// TwinCAT 3 PLC project tcl_Utilities
// Title: tcl_Utilities
// Company: Red Rock Controls Limited
// Author: Roger Christopher
// ProjectVersion: 1.0.9.0
// Description: F_LogError, etc added tcl_EventLog lib ref removed
// ProgramVersion: 3.1.4023.0
// libraries:
//   Tc2_Standard, * (Beckhoff Automation GmbH)
//   Tc2_System, * (Beckhoff Automation GmbH)
//   Tc2_Utilities, * (Beckhoff Automation GmbH)
//   Tc3_Module, * (Beckhoff Automation GmbH)
//   tcl_Events, * (Red Rock Controls Limited)
//   tcl_Execution, * (Red Rock Controls Limited)
//   tcl_UnitTest, * (Red Rock Controls Limited)
// project tree:
//   Classes/Clock/Event Definitions/Day Changed/ IEventHandler_OnDayChanged.TcIO, TEvent_DayChanged.TcPOU
//   Classes/Clock/Event Definitions/Hours Changed/ IEventHandler_OnHourChanged.TcIO, TEvent_HoursChanged.TcPOU
//   Classes/Clock/Event Definitions/Minutes Changed/ IEventHandler_OnMinutesChanged.TcIO, TEvent_MinutesChanged.TcPOU
//   Classes/Clock/Event Definitions/Seconds Changed/ IEventHandler_OnSecondsChanged.TcIO, TEvent_SecondsChanged.TcPOU
//   Classes/Clock/ IClock.TcIO, TClock.TcPOU, TClockEventSource.TcPOU
//   Classes/Edge Detection/ TFallingEdge.TcPOU (not stored), TRisingEdge.TcPOU
//   Classes/Licence Check/ TLicenceCheck.TcPOU
//   Classes/Misc/ TCounter.TcPOU, TCsvString.TcPOU, TGetTimeZoneInfo.TcPOU, TRestartTwinCAT.TcPOU, TRingCounter_INT.TcPOU, TRingCounter_UDINT.TcPOU, TRollingAverage.TcPOU, TSetWindowsClock.TcPOU, TShutdown.TcPOU, TStartProcess.TcPOU
//   Classes/String Split/ TStringSplitter.TcPOU (not stored)
//   Classes/Timers/ TOffTimer.TcPOU (not stored), TOnTimer.TcPOU, TPulseTimer.TcPOU
//   Classes/Value Monitor/ TValueMonitor.TcPOU, TValueMonitorEx.TcPOU
//   Function Blocks/ FB_AutoReset.TcPOU, FB_ValueChanged.TcPOU
//   Functions/Date Time Formatting/ F_DateAsString.TcPOU, F_DateTimeAsString.TcPOU, F_DateTimeAsString_ms.TcPOU, F_TimeAsString.TcPOU, F_TimeAsString_ms.TcPOU, F_TimestampAsFilenameString.TcPOU (not stored)
//   Functions/Event Logging/ F_LogError.TcPOU, F_LogMessage.TcPOU, F_LogWarning.TcPOU
//   Functions/General/ F_ClearMem.TcPOU (not stored), F_GetAdsPort.TcPOU (not stored)
//   Functions/Misc/ F_Assert.TcPOU (not stored), F_Equals.TcPOU (not stored)
//   Functions/String Formatting/ F_FormatString1.TcPOU (not stored), F_FormatString10.TcPOU (not stored), F_FormatString2.TcPOU (not stored), F_FormatString3.TcPOU (not stored), F_FormatString4.TcPOU (not stored), F_FormatString5.TcPOU, F_FormatString6.TcPOU (not stored), F_FormatString7.TcPOU (not stored), F_FormatString8.TcPOU (not stored), F_FormatStringEx1.TcPOU (not stored), F_FormatStringEx10.TcPOU, F_FormatStringEx2.TcPOU (not stored), F_FormatStringEx3.TcPOU (not stored), F_FormatStringEx4.TcPOU (not stored), F_FormatStringEx5.TcPOU (not stored), F_FormatStringEx6.TcPOU, F_FormatStringEx7.TcPOU (not stored), F_FormatStringEx8.TcPOU, F_LREAL_TO_STRING.TcPOU (not stored), F_LTrimEx.TcPOU (not stored), F_PadString.TcPOU, F_RTrimEx.TcPOU, F_STRING_TO_ARG.TcPOU (not stored), F_Trim.TcPOU (not stored)
//   / GlobalTextList.TcGTLO (not stored), Param.TcGVL, PlcTask.TcTTO, Visualization Manager.TcVMO (not stored)
//   Unit Tests/Clock/ Test_Raises_OnDaysChanged.TcPOU, Test_Raises_OnHoursChanged.TcPOU, Test_Raises_OnMinutesChanged.TcPOU, Test_Raises_OnSecondsChanged.TcPOU
//   Unit Tests/Date Time Formatting Tests/ Test_DateAsString.TcPOU, Test_DateTimeAsString.TcPOU, Test_DateTimeAsString_ms.TcPOU, Test_TimeAsString_24HourFormat.TcPOU, Test_TimeAsString_IncludesLeadingZeros.TcPOU, Test_TimestampAsFilenameString.TcPOU, Test_TimeAsString_ms.TcPOU
//   Unit Tests/Licence Check/ Test_LicenceCheck_GetsInValidLicence.TcPOU, Test_LicenceCheck_GetsValidLicence.TcPOU
//   Unit Tests/ PB_TestRunner.TcPOU
//   Unit Tests/String Split/ Test_StringSplitter_Handles_Empty_String.TcPOU, Test_StringSplitter_ReturnsRemainder.TcPOU, Test_StringSplitter_Splits_On_Tab.TcPOU
//   Version/ Global_Version.TcGVL
//   Visualisation/ Visualization.TcVIS
// real-time tasks:
//   TASK PlcTask: cycle T#10ms, priority 20, ADS port 350

CONFIGURATION tcl_Utilities
    RESOURCE PLC ON TwinCAT3
        TASK PlcTask(INTERVAL := T#10ms, PRIORITY := 20);
        PROGRAM PB_TestRunner WITH PlcTask : PB_TestRunner;
    END_RESOURCE
END_CONFIGURATION

// ---- Param.TcGVL
{attribute 'qualified_only'}
VAR_GLOBAL CONSTANT
    MaxCsvFields : INT := 99;
END_VAR

// ---- Version/Global_Version.TcGVL
{attribute 'TcGenerated'}
{attribute 'no-analysis'}
{attribute 'linkalways'}
// This function has been automatically generated from the project information.
VAR_GLOBAL CONSTANT
	{attribute 'const_non_replaced'}
	stLibVersion_tcl_Utilities : ST_LibVersion := (iMajor := 1, iMinor := 0, iBuild := 9, iRevision := 0, nFlags := 0, sVersion := '1.0.9.0');
END_VAR

// ---- Classes/Clock/Event Definitions/Day Changed/IEventHandler_OnDayChanged.TcIO
INTERFACE IEventHandler_OnDayChanged EXTENDS IEventHandlerBase

METHOD OnDayChanged
VAR_INPUT
	Now: TIMESTRUCT;
END_VAR
END_METHOD

END_INTERFACE

// ---- Classes/Clock/Event Definitions/Hours Changed/IEventHandler_OnHourChanged.TcIO
INTERFACE IEventHandler_OnHourChanged EXTENDS IEventHandlerBase

METHOD OnHourChanged
VAR_INPUT
	Now: TIMESTRUCT;
END_VAR
END_METHOD

END_INTERFACE

// ---- Classes/Clock/Event Definitions/Minutes Changed/IEventHandler_OnMinutesChanged.TcIO
INTERFACE IEventHandler_OnMinutesChanged EXTENDS IEventHandlerBase

METHOD OnMinutesChanged
VAR_INPUT
	Now: TIMESTRUCT;
END_VAR
END_METHOD

END_INTERFACE

// ---- Classes/Clock/Event Definitions/Seconds Changed/IEventHandler_OnSecondsChanged.TcIO
INTERFACE IEventHandler_OnSecondsChanged EXTENDS IEventHandlerBase

METHOD OnSecondsChanged
VAR_INPUT
	Now: TIMESTRUCT;
END_VAR
END_METHOD

END_INTERFACE

// ---- Classes/Clock/IClock.TcIO
INTERFACE IClock

PROPERTY DateTimeInitialised : BOOL
GET
END_GET
END_PROPERTY

PROPERTY NowAsDateTime : DT
GET
END_GET
END_PROPERTY

PROPERTY NowAsTimeStruct : REFERENCE TO TIMESTRUCT
GET
END_GET
END_PROPERTY

END_INTERFACE

// ---- Unit Tests/PB_TestRunner.TcPOU
PROGRAM PB_TestRunner 
VAR
//    EnableAdsLogMessages_State : BOOL;
//    EnableAdsLogMessages_DuringTest : BOOL := FALSE; // inhibit Invalid Event Handler error message - confusing here
//    RisingEdge_TestsRunning  : TRisingEdge;
//    FallingEdge_TestsRunning : TFallingEdge;
    
    Test_Raises_OnDaysChanged                : Test_Raises_OnDaysChanged;
    Test_Raises_OnHoursChanged               : Test_Raises_OnHoursChanged;
    Test_Raises_OnMinutesChanged             : Test_Raises_OnMinutesChanged;
    Test_Raises_OnSecondsChanged             : Test_Raises_OnSecondsChanged;
                                             
    Test_DateAsString                        : Test_DateAsString;
    Test_DateTimeAsString                    : Test_DateTimeAsString;
    Test_DateTimeAsString_ms                 : Test_DateTimeAsString_ms;
    Test_TimeAsString_24HourFormat           : Test_TimeAsString_24HourFormat;
    Test_TimeAsString_IncludesLeadingZeros   : Test_TimeAsString_IncludesLeadingZeros;
    Test_TimeAsString_ms                     : Test_TimeAsString_ms;
    Test_TimestampAsFilenameString           : Test_TimestampAsFilenameString;
                                             
    Test_LicenceCheck_GetsInValidLicence     : Test_LicenceCheck_GetsInValidLicence;
    Test_LicenceCheck_GetsValidLicence       : Test_LicenceCheck_GetsValidLicence;
   
    Test_StringSplitter_Handles_Empty_String : Test_StringSplitter_Handles_Empty_String;
    Test_StringSplitter_ReturnsRemainder     : Test_StringSplitter_ReturnsRemainder;
    Test_StringSplitter_Splits_On_Tab        : Test_StringSplitter_Splits_On_Tab;

 
END_VAR

tcl_UnitTest.TestFramework.TestRunner();

//IF RisingEdge_TestsRunning.Test(tcl_UnitTest.UnitTests.TestFramework.TestsRunning) THEN
//    EnableAdsLogMessages_State := tcl_EventLog.EventLog.EnableAdsLogMessages; // store so we can restore previous state
//    EventLog.EnableAdsLogMessages := EnableAdsLogMessages_DuringTest;  // force the visibility of ads log messages
//END_IF

//IF FallingEdge_TestsRunning.Test(tcl_UnitTest.UnitTests.TestFramework.TestsRunning) THEN
//    EventLog.EnableAdsLogMessages := EnableAdsLogMessages_State; // restore previous state
//END_IF

END_PROGRAM

// ---- Unit Tests/Clock/Test_Raises_OnDaysChanged.TcPOU
FUNCTION_BLOCK Test_Raises_OnDaysChanged EXTENDS TUnitTestBase
IMPLEMENTS 
    IEventHandler_OnDayChanged
VAR
    NowFromEvent : TIMESTRUCT;
    
    OnDaysChanged_Raised    : BOOL;
END_VAR

METHOD  Execute
VAR_INST
    ClockEventSource : TClockEventSource;
    Now              : TIMESTRUCT := (wDay := 23, wMonth := 12, wYear := 1945, wHour := 22, wMinute := 20, wSecond := 18);
    OneDayLater      : TIMESTRUCT := (wDay := 24, wMonth := 12, wYear := 1945, wHour := 22, wMinute := 20, wSecond := 18);
END_VAR
OnDaysChanged_Raised := FALSE;

ClockEventSource.Event_DayChanged.ClearEventHandlers().AddEventHandler(THIS^);

ClockEventSource.Init(Now := Now);
ClockEventSource(Now := OneDayLater);

Assertion.AssertEquals_BOOL(
    Expected := TRUE,
    Actual   := OnDaysChanged_Raised,
    ObjectName := _TestName,
    VariableName  := 'OnDaysChanged_Raised');

Assertion.AssertEquals_STRUCT(
    Expected := OneDayLater,
    Actual   := NowFromEvent,
    ObjectName := _TestName,
    VariableName  := 'NowFromEvent');

Test_Finished();
END_METHOD

METHOD OnDayChanged
VAR_INPUT
	Now	: Tc2_Utilities.TIMESTRUCT;
END_VAR
NowFromEvent := Now;
OnDaysChanged_Raised := TRUE;
END_METHOD

END_FUNCTION_BLOCK

// ---- Classes/Clock/TClockEventSource.TcPOU
FUNCTION_BLOCK TClockEventSource
VAR_INPUT
    Now : TIMESTRUCT;
END_VAR
VAR
    _LastTickNowAsTimestruct : TIMESTRUCT;

    _Event_SecondsChanged : TEvent_SecondsChanged;
    _Event_MinutesChanged : TEvent_MinutesChanged;
    _Event_HoursChanged   : TEvent_HoursChanged;
    _Event_DayChanged     : TEvent_DayChanged;

END_VAR

IF Now.wSecond <> _LastTickNowAsTimestruct.wSecond THEN
    _Event_SecondsChanged.RaiseEx(Now);
END_IF
IF Now.wMinute <> _LastTickNowAsTimestruct.wMinute THEN
    _Event_MinutesChanged.RaiseEx(Now);
END_IF
IF Now.wHour <> _LastTickNowAsTimestruct.wHour THEN
    _Event_HoursChanged.RaiseEx(Now);
END_IF
IF Now.wDay <> _LastTickNowAsTimestruct.wDay THEN
    _Event_DayChanged.RaiseEx(Now);
END_IF

_LastTickNowAsTimestruct := Now;

PROPERTY Event_DayChanged : IEvent
GET
Event_DayChanged := _Event_DayChanged;
END_GET
END_PROPERTY

PROPERTY Event_HoursChanged : IEvent
GET
Event_HoursChanged := _Event_HoursChanged;
END_GET
END_PROPERTY

PROPERTY Event_MinutesChanged : IEvent
GET
Event_MinutesChanged := _Event_MinutesChanged;
END_GET
END_PROPERTY

PROPERTY Event_SecondsChanged : IEvent
GET
Event_SecondsChanged := _Event_SecondsChanged;
END_GET
END_PROPERTY

METHOD Init // initialise stored value so event handlers do not fire erroneously on first update
VAR_INPUT
    Now : TIMESTRUCT;
END_VAR
_LastTickNowAsTimestruct := Now;
END_METHOD

END_FUNCTION_BLOCK

// ---- Classes/Clock/Event Definitions/Seconds Changed/TEvent_SecondsChanged.TcPOU
FUNCTION_BLOCK TEvent_SecondsChanged EXTENDS TEventBase IMPLEMENTS IEvent
VAR
	Now: TIMESTRUCT;
    Handler : IEventHandler_OnSecondsChanged;
END_VAR

METHOD  CallHandler
VAR_INPUT
    HandlerBase : IEventHandlerBase;
END_VAR
IF __QUERYINTERFACE(HandlerBase,Handler) THEN
    Handler.OnSecondsChanged(Now);
END_IF
END_METHOD

METHOD  IsHandlerSupported : BOOL
VAR_INPUT
    EventHandler : IEventHandlerBase;
END_VAR
IF __QUERYINTERFACE(EventHandler,Handler) THEN
    IsHandlerSupported := TRUE;
END_IF
END_METHOD

METHOD RaiseEx
VAR_INPUT
	Now: TIMESTRUCT;
END_VAR
THIS^.Now := Now;
SUPER^.Raise();
END_METHOD

END_FUNCTION_BLOCK

// ---- Classes/Clock/Event Definitions/Minutes Changed/TEvent_MinutesChanged.TcPOU
FUNCTION_BLOCK TEvent_MinutesChanged EXTENDS TEventBase IMPLEMENTS IEvent
VAR
	Now: TIMESTRUCT;
    Handler : IEventHandler_OnMinutesChanged;
END_VAR

METHOD  CallHandler
VAR_INPUT
    HandlerBase : IEventHandlerBase;
END_VAR
IF __QUERYINTERFACE(HandlerBase,Handler) THEN
    Handler.OnMinutesChanged(Now);
END_IF
END_METHOD

METHOD  IsHandlerSupported : BOOL
VAR_INPUT
    EventHandler : IEventHandlerBase;
END_VAR
IF __QUERYINTERFACE(EventHandler,Handler) THEN
    IsHandlerSupported := TRUE;
END_IF
END_METHOD

METHOD RaiseEx
VAR_INPUT
	Now: TIMESTRUCT;
END_VAR
THIS^.Now := Now;
SUPER^.Raise();
END_METHOD

END_FUNCTION_BLOCK

// ---- Classes/Clock/Event Definitions/Hours Changed/TEvent_HoursChanged.TcPOU
FUNCTION_BLOCK TEvent_HoursChanged EXTENDS TEventBase IMPLEMENTS IEvent
VAR
	Now: TIMESTRUCT;
    Handler : IEventHandler_OnHourChanged;
END_VAR

METHOD  CallHandler
VAR_INPUT
    HandlerBase : IEventHandlerBase;
END_VAR
IF __QUERYINTERFACE(HandlerBase,Handler) THEN
    Handler.OnHourChanged(Now);
END_IF
END_METHOD

METHOD  IsHandlerSupported : BOOL
VAR_INPUT
    EventHandler : IEventHandlerBase;
END_VAR
IF __QUERYINTERFACE(EventHandler,Handler) THEN
    IsHandlerSupported := TRUE;
END_IF
END_METHOD

METHOD RaiseEx
VAR_INPUT
	Now: TIMESTRUCT;
END_VAR
THIS^.Now := Now;
SUPER^.Raise();
END_METHOD

END_FUNCTION_BLOCK

// ---- Classes/Clock/Event Definitions/Day Changed/TEvent_DayChanged.TcPOU
FUNCTION_BLOCK TEvent_DayChanged EXTENDS TEventBase IMPLEMENTS IEvent
VAR
	Now: TIMESTRUCT;
    Handler : IEventHandler_OnDayChanged;
END_VAR

METHOD  CallHandler
VAR_INPUT
    HandlerBase : IEventHandlerBase;
END_VAR
IF __QUERYINTERFACE(HandlerBase,Handler) THEN
    Handler.OnDayChanged(Now);
END_IF
END_METHOD

METHOD  IsHandlerSupported : BOOL
VAR_INPUT
    EventHandler : IEventHandlerBase;
END_VAR
IF __QUERYINTERFACE(EventHandler,Handler) THEN
    IsHandlerSupported := TRUE;
END_IF
END_METHOD

METHOD RaiseEx
VAR_INPUT
	Now: TIMESTRUCT;
END_VAR
THIS^.Now := Now;
SUPER^.Raise();
END_METHOD

END_FUNCTION_BLOCK

// ---- Unit Tests/Clock/Test_Raises_OnHoursChanged.TcPOU
FUNCTION_BLOCK Test_Raises_OnHoursChanged EXTENDS TUnitTestBase
IMPLEMENTS 
    IEventHandler_OnHourChanged
VAR
    NowFromEvent : TIMESTRUCT;
    
    OnHoursChanged_Raised    : BOOL;
END_VAR

METHOD  Execute
VAR_INST
    ClockEventSource : TClockEventSource;
    Now              : TIMESTRUCT := (wDay := 23, wMonth := 12, wYear := 1945, wHour := 22, wMinute := 20, wSecond := 18);
    OneHourLater     : TIMESTRUCT := (wDay := 23, wMonth := 12, wYear := 1945, wHour := 23, wMinute := 20, wSecond := 18);
END_VAR
OnHoursChanged_Raised := FALSE;

ClockEventSource.Event_HoursChanged.ClearEventHandlers().AddEventHandler(THIS^);

ClockEventSource.Init(Now := Now);
ClockEventSource(Now := OneHourLater);

Assertion.AssertEquals_BOOL(
    Expected := TRUE,
    Actual   := OnHoursChanged_Raised,
    ObjectName := _TestName,
    VariableName  := 'OnHoursChanged_Raised');

Assertion.AssertEquals_STRUCT(
    Expected := OneHourLater,
    Actual   := NowFromEvent,
    ObjectName := _TestName,
    VariableName  := 'NowFromEvent');

Test_Finished();
END_METHOD

METHOD OnHourChanged
VAR_INPUT
	Now	: Tc2_Utilities.TIMESTRUCT;
END_VAR
NowFromEvent := Now;
OnHoursChanged_Raised := TRUE;
END_METHOD

END_FUNCTION_BLOCK

// ---- Unit Tests/Clock/Test_Raises_OnMinutesChanged.TcPOU
FUNCTION_BLOCK Test_Raises_OnMinutesChanged EXTENDS TUnitTestBase
IMPLEMENTS 
    IEventHandler_OnMinutesChanged
VAR
    NowFromEvent : TIMESTRUCT;
    
    OnMinutesChanged_Raised    : BOOL;
END_VAR

METHOD  Execute
VAR_INST
    ClockEventSource : TClockEventSource;
    Now              : TIMESTRUCT := (wDay := 23, wMonth := 12, wYear := 1945, wHour := 22, wMinute := 20, wSecond := 18);
    OneMinuteLater   : TIMESTRUCT := (wDay := 23, wMonth := 12, wYear := 1945, wHour := 22, wMinute := 21, wSecond := 18);
END_VAR
OnMinutesChanged_Raised := FALSE;

ClockEventSource.Event_MinutesChanged.ClearEventHandlers().AddEventHandler(THIS^);

ClockEventSource.Init(Now := Now);
ClockEventSource(Now := OneMinuteLater);

Assertion.AssertEquals_BOOL(
    Expected := TRUE,
    Actual   := OnMinutesChanged_Raised,
    ObjectName := _TestName,
    VariableName  := 'OnMinutesChanged_Raised');

Assertion.AssertEquals_STRUCT(
    Expected := OneMinuteLater,
    Actual   := NowFromEvent,
    ObjectName := _TestName,
    VariableName  := 'NowFromEvent');

Test_Finished();
END_METHOD

METHOD OnMinutesChanged
VAR_INPUT
	Now	: Tc2_Utilities.TIMESTRUCT;
END_VAR
NowFromEvent := Now;
OnMinutesChanged_Raised := TRUE;
END_METHOD

END_FUNCTION_BLOCK

// ---- Unit Tests/Clock/Test_Raises_OnSecondsChanged.TcPOU
FUNCTION_BLOCK Test_Raises_OnSecondsChanged EXTENDS TUnitTestBase
IMPLEMENTS 
    IEventHandler_OnSecondsChanged
VAR
    NowFromEvent : TIMESTRUCT;
    
    OnSecondsChanged_Raised    : BOOL;
END_VAR

METHOD  Execute
VAR_INST
    ClockEventSource : TClockEventSource;
    Now              : TIMESTRUCT := (wDay := 23, wMonth := 12, wYear := 1945, wHour := 22, wMinute := 20, wSecond := 18);
    OneSecondLater   : TIMESTRUCT := (wDay := 23, wMonth := 12, wYear := 1945, wHour := 22, wMinute := 20, wSecond := 19);
END_VAR
OnSecondsChanged_Raised := FALSE;

ClockEventSource.Event_SecondsChanged.ClearEventHandlers().AddEventHandler(THIS^);

ClockEventSource.Init(Now := Now);
ClockEventSource(Now := OneSecondLater);

Assertion.AssertEquals_BOOL(
    Expected := TRUE,
    Actual   := OnSecondsChanged_Raised,
    ObjectName := _TestName,
    VariableName  := 'OnSecondsChanged_Raised');

Assertion.AssertEquals_STRUCT(
    Expected := OneSecondLater,
    Actual   := NowFromEvent,
    ObjectName := _TestName,
    VariableName  := 'NowFromEvent');

Test_Finished();
END_METHOD

METHOD OnSecondsChanged
VAR_INPUT
	Now	: Tc2_Utilities.TIMESTRUCT;
END_VAR
NowFromEvent := Now;
OnSecondsChanged_Raised := TRUE;
END_METHOD

END_FUNCTION_BLOCK

// ---- Unit Tests/Date Time Formatting Tests/Test_DateAsString.TcPOU
FUNCTION_BLOCK Test_DateAsString EXTENDS TUnitTestBase
VAR
END_VAR

METHOD  Execute
VAR_INST
    TimeStruct : TIMESTRUCT := (wDay := 23, wMonth := 12, wYear := 1945);
END_VAR
Assertion.AssertEquals_STRING(
    Expected := '23/12/1945',
    Actual   := F_DateAsString(TimeStruct),
    ObjectName := _TestName,
    VariableName  := 'F_DateAsString(TimeStruct)');


Test_Finished();
END_METHOD

END_FUNCTION_BLOCK

// ---- Functions/Date Time Formatting/F_DateAsString.TcPOU
FUNCTION F_DateAsString : T_MaxString
VAR_INPUT
    TimeStruct : TIMESTRUCT;
END_VAR

F_DateAsString := F_FormatString3(
                      Format := '%.2d/%.2d/%.2d',
                      arg1   := F_WORD(TimeStruct.wDay),
                      arg2   := F_WORD(TimeStruct.wMonth),
                      arg3   := F_WORD(TimeStruct.wYear));

END_FUNCTION

// ---- Unit Tests/Date Time Formatting Tests/Test_DateTimeAsString.TcPOU
FUNCTION_BLOCK Test_DateTimeAsString EXTENDS TUnitTestBase
VAR
END_VAR

METHOD  Execute
VAR_INST
    TimeStruct : TIMESTRUCT := (wDay := 23, wMonth := 12, wYear := 1945, wHour := 22, wMinute := 20, wSecond := 18);
END_VAR
AssertEquals_STRING(
    Expected := '22:20:18 23/12/1945',
    Actual   := F_DateTimeAsString(TimeStruct),
    VariableName  := 'F_DateTimeAsString(TimeStruct)');


Test_Finished();
END_METHOD

END_FUNCTION_BLOCK

// ---- Functions/Date Time Formatting/F_DateTimeAsString.TcPOU
FUNCTION F_DateTimeAsString : T_MaxString
VAR_INPUT
    TimeStruct : TIMESTRUCT;
END_VAR

F_DateTimeAsString := F_FormatStringEx2(
                          Format := '%s %s',
                          arg1   := F_TimeAsString(TimeStruct),
                          arg2   := F_DateAsString(TimeStruct));

END_FUNCTION

// ---- Functions/Date Time Formatting/F_TimeAsString.TcPOU
FUNCTION F_TimeAsString : T_MaxString
VAR_INPUT
    TimeStruct : TIMESTRUCT;
END_VAR

F_TimeAsString := F_FormatString3(
                      Format := '%.2d:%.2d:%.2d',
                      arg1   := F_WORD(TimeStruct.wHour),
                      arg2   := F_WORD(TimeStruct.wMinute),
                      arg3   := F_WORD(TimeStruct.wSecond));

END_FUNCTION

// ---- Unit Tests/Date Time Formatting Tests/Test_DateTimeAsString_ms.TcPOU
FUNCTION_BLOCK Test_DateTimeAsString_ms EXTENDS TUnitTestBase
VAR
END_VAR

METHOD  Execute
VAR_INST
    TimeStruct : TIMESTRUCT := (wDay := 23, wMonth := 12, wYear := 1945, wHour := 22, wMinute := 20, wSecond := 18, wMilliseconds := 512);
END_VAR
AssertEquals_STRING(
    Expected := '22:20:18.512 23/12/1945',
    Actual   := F_DateTimeAsString_ms(TimeStruct),
    VariableName  := 'F_DateTimeAsString_ms(TimeStruct)');


Test_Finished();
END_METHOD

END_FUNCTION_BLOCK

// ---- Functions/Date Time Formatting/F_DateTimeAsString_ms.TcPOU
FUNCTION F_DateTimeAsString_ms : T_MaxString
VAR_INPUT
    TimeStruct : TIMESTRUCT;
END_VAR
VAR
	FB_FormatString1 : FB_FormatString;
END_VAR

F_DateTimeAsString_ms := F_FormatStringEx2(
                             Format := '%s %s',
                             arg1   := F_TimeAsString_ms(TimeStruct),
                             arg2   := F_DateAsString(TimeStruct));

END_FUNCTION

// ---- Functions/Date Time Formatting/F_TimeAsString_ms.TcPOU
FUNCTION F_TimeAsString_ms : T_MaxString
VAR_INPUT
    TimeStruct : TIMESTRUCT;
END_VAR

F_TimeAsString_ms := F_FormatString4(
                         Format := '%.2d:%.2d:%.2d.%.3d',
                         arg1   := F_WORD(TimeStruct.wHour),
                         arg2   := F_WORD(TimeStruct.wMinute),
                         arg3   := F_WORD(TimeStruct.wSecond),
   	                     arg4   := F_WORD(TimeStruct.wMilliseconds));

END_FUNCTION

// ---- Unit Tests/Date Time Formatting Tests/Test_TimeAsString_24HourFormat.TcPOU
FUNCTION_BLOCK Test_TimeAsString_24HourFormat EXTENDS TUnitTestBase
VAR
END_VAR

METHOD  Execute
VAR_INST
    TimeStruct : TIMESTRUCT := (wHour := 22, wMinute := 20, wSecond := 18);
END_VAR
Assertion.AssertEquals_STRING(
    Expected := '22:20:18',
    Actual   := F_TimeAsString(TimeStruct),
    ObjectName := _TestName,
    VariableName  := 'F_TimeAsString(TimeStruct)');


Test_Finished();
END_METHOD

END_FUNCTION_BLOCK

// ---- Unit Tests/Date Time Formatting Tests/Test_TimeAsString_IncludesLeadingZeros.TcPOU
FUNCTION_BLOCK Test_TimeAsString_IncludesLeadingZeros EXTENDS TUnitTestBase
VAR
END_VAR

METHOD  Execute
VAR_INST
    TimeStruct : TIMESTRUCT := (wHour := 6, wMinute := 5, wSecond := 4);
END_VAR
Assertion.AssertEquals_STRING(
    Expected := '06:05:04',
    Actual   := F_TimeAsString(TimeStruct),
    ObjectName := _TestName,
    VariableName  := 'F_TimeAsString(TimeStruct)');


Test_Finished();
END_METHOD

END_FUNCTION_BLOCK

// ---- Unit Tests/Date Time Formatting Tests/Test_TimeAsString_ms.TcPOU
FUNCTION_BLOCK Test_TimeAsString_ms EXTENDS TUnitTestBase
VAR
END_VAR

METHOD  Execute
VAR_INST
    TimeStruct : TIMESTRUCT := (wHour := 6, wMinute := 5, wSecond := 4, wMilliseconds := 135);
END_VAR
Assertion.AssertEquals_STRING(
    Expected := '06:05:04.135',
    Actual   := F_TimeAsString_ms(TimeStruct),
    ObjectName := _TestName,
    VariableName  := 'F_TimeAsString_ms(TimeStruct)');


Test_Finished();
END_METHOD

END_FUNCTION_BLOCK

// ---- Unit Tests/Date Time Formatting Tests/Test_TimestampAsFilenameString.TcPOU
FUNCTION_BLOCK Test_TimestampAsFilenameString EXTENDS TUnitTestBase
VAR
END_VAR

METHOD  Execute
VAR_INST
    TimeStruct : TIMESTRUCT := (wDay := 23, wMonth := 12, wYear := 1945, wHour := 22, wMinute := 20, wSecond := 18, wMilliseconds := 512);
END_VAR
AssertEquals_STRING(
    Expected := '1945-12-23 22-20-18',
    Actual   := F_TimestampAsFilenameString(TimeStruct),
    VariableName  := 'F_TimeAsString_ms(TimeStruct)');


Test_Finished();
END_METHOD

END_FUNCTION_BLOCK

// ---- Unit Tests/Licence Check/Test_LicenceCheck_GetsInValidLicence.TcPOU
FUNCTION_BLOCK Test_LicenceCheck_GetsInValidLicence EXTENDS TUnitTestBase
VAR
END_VAR

METHOD  Execute
VAR_INST
    LicenceCheck : TLicenceCheck(
        LicenceIdAsString      := '{13ae39d9-bbb2-423e-8ace-d2c791a6b0ec}', // 1st digit should be 0
        LicenceName            := 'tcl_BaseLib',
        StopTwinCAT_IfNotValid := FALSE);
END_VAR
IF NOT TestStarted THEN
    LicenceCheck.FB_init(
        bInitRetains            := FALSE,
        bInCopyCode             := FALSE,
        LicenceIdAsString      := '{13ae39d9-bbb2-423e-8ace-d2c791a6b0ec}', // 1st digit should be 0
        LicenceName            := 'tcl_BaseLib',
        StopTwinCAT_IfNotValid := FALSE);
    Test_Started();
END_IF
LicenceCheck();

IF LicenceCheck.CheckComplete THEN
    Assertion.AssertEquals_BOOL(
        Expected := FALSE,
        Actual   := LicenceCheck.IsValid,
        ObjectName := _TestName,
        VariableName  := 'LicenceCheck.IsValid');
    Test_Finished();
END_IF
END_METHOD

END_FUNCTION_BLOCK

// ---- Classes/Licence Check/TLicenceCheck.TcPOU
FUNCTION_BLOCK TLicenceCheck
VAR
    LicenceIdAsString : STRING(38);
    LicenceName : T_MaxString;
    StopTwinCAT_IfNotValid : BOOL;

    FB_GetLicenses1 : FB_GetLicenses;
    FallingEdge_Busy : TFallingEdge;
    ScanCount : UDINT;
    OnTimer_CheckComplete : TOnTimer(PresetTime := 0.1);
    StopTwinCAT : TC_Stop;
    LicenceId : GUID;
    i : UDINT;
    
    _IsValid : BOOL;
    _CheckComplete : BOOL;
    _StopTwinCAT : BOOL;
END_VAR

IF _IsValid THEN
    RETURN;
END_IF

ScanCount := ScanCount + 1;

FB_GetLicenses1(
	bExecute:= TRUE, 
	tTimeout:= , 
	sNetId:= , 
	bBusy=> , 
	bError=> , 
	nErrorId=> , 
	nValidLicenses=> , 
	aValidLicenses=> , 
	nInvalidLicenses=> , 
	aInvalidLicenses=> );

IF FallingEdge_Busy.Test(FB_GetLicenses1.bBusy) THEN
    _CheckComplete := TRUE;
    IF FB_GetLicenses1.bError THEN
            F_LogError('Licence Check',F_FormatString1('Error %X retrieving TwinCAT licences',F_UDINT(FB_GetLicenses1.nErrorId)));
    ELSE
        IF FB_GetLicenses1.nValidLicenses > 0 THEN
            LicenceId := REGSTRING_TO_GUID(LicenceIdAsString);
            FOR i := 1 TO FB_GetLicenses1.nValidLicenses DO
                IF GuidsEqualByVal(FB_GetLicenses1.aValidLicenses[i].stLicenseId, LicenceId) THEN
                    _IsValid := TRUE;
                END_IF
            END_FOR
        END_IF	
    END_IF
    IF NOT _IsValid THEN
        IF StopTwinCAT_IfNotValid THEN
            F_LogError('Licence Check',F_FormatStringEx2('Licence "%s" with ID %s not found: TwinCAT will be stopped!',LicenceName,LicenceIdAsString));
            ScanCount := 0;
            OnTimer_CheckComplete.Run();
            _StopTwinCAT := TRUE;
        ELSE
            F_LogError('Licence Check',F_FormatStringEx2('Licence "%s" with ID %s not found.',LicenceName,LicenceIdAsString));
		END_IF
    END_IF
END_IF

IF _StopTwinCAT THEN
    IF ScanCount > 5 OR OnTimer_CheckComplete.Run() THEN // scan count used when cyclically executed, timer used where executed sporadically
        StopTwinCAT(
            NETID:= , 
            STOP:= TRUE, 
            TMOUT:= , 
            BUSY=> , 
            ERR=> , 
            ERRID=> );
	END_IF
END_IF

PROPERTY CheckComplete : BOOL
GET
CheckComplete := _CheckComplete;
END_GET
END_PROPERTY

METHOD FB_init : BOOL
VAR_INPUT
	bInitRetains : BOOL; // if TRUE, the retain variables are initialized (warm start / cold start)
	bInCopyCode : BOOL;  // if TRUE, the instance afterwards gets moved into the copy code (online change)
    LicenceIdAsString : STRING(38);
    LicenceName : T_MaxString;
    StopTwinCAT_IfNotValid : BOOL;
END_VAR
THIS^.LicenceIdAsString         := LicenceIdAsString;
THIS^.LicenceName               := LicenceName;
THIS^.StopTwinCAT_IfNotValid    := StopTwinCAT_IfNotValid;
THIS^._IsValid                  := FALSE;
THIS^._CheckComplete            := FALSE;
END_METHOD

PROPERTY IsValid : BOOL
GET
IsValid := _IsValid;
END_GET
END_PROPERTY

END_FUNCTION_BLOCK

// ---- Classes/Timers/TOnTimer.TcPOU
FUNCTION_BLOCK TOnTimer
VAR
    TON1 : TON;
END_VAR

METHOD Delay : BOOL
VAR_INPUT
    In : BOOL;
END_VAR
TON1(IN := In);
Delay := TON1.Q;
END_METHOD

METHOD FB_init : BOOL
VAR_INPUT
	bInitRetains : BOOL; // if TRUE, the retain variables are initialized (warm start / cold start)
	bInCopyCode : BOOL;  // if TRUE, the instance afterwards gets moved into the copy code (online change)
    PresetTime : LREAL; // seconds
END_VAR
TON1.PT := LREAL_TO_TIME(PresetTime * 1000);
END_METHOD

PROPERTY OutputState : BOOL
GET
OutputState := TON1.Q;
END_GET
END_PROPERTY

PROPERTY PresetTime : LREAL
GET
PresetTime := TIME_TO_LREAL(TON1.PT)/1000.0; // in seconds
END_GET
SET
TON1.PT := LREAL_TO_TIME(PresetTime * 1000);
END_SET
END_PROPERTY

METHOD Reset
TON1(IN := FALSE);
END_METHOD

METHOD Run : BOOL
TON1(IN := TRUE);
Run := TON1.Q;
END_METHOD

END_FUNCTION_BLOCK

// ---- Functions/Event Logging/F_LogError.TcPOU
FUNCTION F_LogError  
VAR_INPUT
    Source  : T_MaxString;
    Message : T_MaxString;
END_VAR

ADSLOGSTR(
        msgCtrlMask := ADSLOG_MSGTYPE_STRING OR ADSLOG_MSGTYPE_ERROR OR ADSLOG_MSGTYPE_LOG,
        msgFmtStr := F_FormatStringEx2('%s : %s',Source,Message),
        strArg := '');

END_FUNCTION

// ---- Unit Tests/Licence Check/Test_LicenceCheck_GetsValidLicence.TcPOU
FUNCTION_BLOCK Test_LicenceCheck_GetsValidLicence EXTENDS TUnitTestBase
VAR
END_VAR

METHOD  Execute
VAR_INST
    LicenceCheck : TLicenceCheck(
        LicenceIdAsString      := '{4c256767-e6e6-4af5-bd68-9f7abad0c200}', // Tc_Ads Id
        LicenceName            := 'Tc_Ads',
        StopTwinCAT_IfNotValid := FALSE);
END_VAR
IF NOT TestStarted THEN
    LicenceCheck.FB_init(
        bInitRetains            := FALSE,
        bInCopyCode             := FALSE,
        LicenceIdAsString      := '{4c256767-e6e6-4af5-bd68-9f7abad0c200}', // 1st digit should be 0
        LicenceName            := 'Tc_Ads',
        StopTwinCAT_IfNotValid := FALSE);
    Test_Started();
END_IF
LicenceCheck();

IF LicenceCheck.CheckComplete THEN
    Assertion.AssertEquals_BOOL(
        Expected := TRUE,
        Actual   := LicenceCheck.IsValid,
        ObjectName := _TestName,
        VariableName  := 'LicenceCheck.IsValid');
    Test_Finished();
END_IF
END_METHOD

END_FUNCTION_BLOCK

// ---- Unit Tests/String Split/Test_StringSplitter_Handles_Empty_String.TcPOU
FUNCTION_BLOCK Test_StringSplitter_Handles_Empty_String EXTENDS TUnitTestBase
VAR
END_VAR

METHOD  Execute
VAR_INST
    StringSplitter : TStringSplitter;
END_VAR
Test_Started();

StringSplitter.Init(
    Str    := '',
    Delim1 := '$T',
    Delim2 := '');

Assertion.AssertEquals_STRING(
    Expected := '',
    Actual   := StringSplitter.GetNext(),
    ObjectName := _TestName,
    VariableName  := 'StringSplitter.GetNext()');

Assertion.AssertEquals_BOOL(
    Expected := FALSE,
    Actual   := StringSplitter.HasMore(),
    ObjectName := _TestName,
    VariableName  := 'StringSplitter.HasMore()');


Test_Finished();
END_METHOD

END_FUNCTION_BLOCK

// ---- Unit Tests/String Split/Test_StringSplitter_ReturnsRemainder.TcPOU
FUNCTION_BLOCK Test_StringSplitter_ReturnsRemainder EXTENDS TUnitTestBase
VAR
END_VAR

METHOD  Execute
VAR_INST
    StringSplitter : TStringSplitter;
END_VAR
Test_Started();

StringSplitter.Init(
    Str    := 'Bob$TCharles$TDavid',
    Delim1 := '$T',
    Delim2 := '');

AssertEquals_BOOL(
    Expected := TRUE,
    Actual   := StringSplitter.HasMore(),
    VariableName  := 'StringSplitter.HasMore()');
    
AssertEquals_STRING(
    Expected := 'Bob',
    Actual   := StringSplitter.GetNext(),
    VariableName  := 'StringSplitter.GetNext()');
    
AssertEquals_STRING(
    Expected := 'Charles$TDavid',
    Actual   := StringSplitter.GetRemainder(),
    VariableName  := 'StringSplitter.GetRemainder()');

AssertEquals_STRING(
    Expected := '',
    Actual   := StringSplitter.GetRemainder(),
    VariableName  := 'StringSplitter.GetRemainder()');

AssertEquals_BOOL(
    Expected := FALSE,
    Actual   := StringSplitter.HasMore(),
    VariableName  := 'StringSplitter.HasMore()');
    

Test_Finished();
END_METHOD

END_FUNCTION_BLOCK

// ---- Unit Tests/String Split/Test_StringSplitter_Splits_On_Tab.TcPOU
FUNCTION_BLOCK Test_StringSplitter_Splits_On_Tab EXTENDS TUnitTestBase
VAR
END_VAR

METHOD  Execute
VAR_INST
    StringSplitter : TStringSplitter;
END_VAR
Test_Started();

StringSplitter.Init(
    Str    := 'Bob$TCharles$TDavid',
    Delim1 := '$T',
    Delim2 := '');

AssertEquals_STRING(
    Expected := 'Bob',
    Actual   := StringSplitter.GetNext(),
    VariableName  := 'StringSplitter.GetNext()');

AssertEquals_STRING(
    Expected := 'Charles',
    Actual   := StringSplitter.GetNext(),
    VariableName  := 'StringSplitter.GetNext()');

AssertEquals_STRING(
    Expected := 'David',
    Actual   := StringSplitter.GetNext(),
    VariableName  := 'StringSplitter.GetNext()');


Test_Finished();
END_METHOD

END_FUNCTION_BLOCK

// ---- Classes/Clock/TClock.TcPOU
FUNCTION_BLOCK TClock IMPLEMENTS IClock
VAR
    _DateTimeInitialised : BOOL; // to detect startup
	_NowAsTimeStruct: TIMESTRUCT;
    
	NT_GetTime1: NT_GetTime;
	TON1: TON;
    GetWindowsTimeRequest : BOOL;
	SyncRequest: BOOL;
    F_TRIG1 : F_TRIG;
	RTC_EX2: RTC_EX2;
	PresetTime: TIMESTRUCT;
    
END_VAR

// Request a sync every 10s
TON1(IN := NOT GetWindowsTimeRequest, PT := T#10S, Q=> GetWindowsTimeRequest);

// Get time from Windows clock
NT_GetTime1(
	NetId := '',
	Start := GetWindowsTimeRequest OR NOT _DateTimeInitialised, // request on first scan also
	TmOut := T#2S,
    Busy => ,
    Err => ,
    ErrId => ,
	TimeStr => PresetTime);

// Request sync to Windows time when time received
F_TRIG1(CLK :=  NT_GetTime1.Busy, Q=> SyncRequest);   
    
// Sync RTC to Windows time
RTC_EX2(
	EN:= SyncRequest, // re-initialise to Windows clock following sync request
	PDT:= PresetTime, // time to sync to
	PMICRO:= PresetTime.wMilliseconds, 
	Q=> , 
	CDT=> _NowAsTimeStruct, // time updated on every call
	CMICRO=> );
    
IF SyncRequest THEN    
    _DateTimeInitialised := TRUE;
END_IF

PROPERTY DateTimeInitialised : BOOL
GET
DateTimeInitialised := _DateTimeInitialised;
END_GET
END_PROPERTY

PROPERTY NowAsDateTime : DT
GET
NowAsDateTime := SYSTEMTIME_TO_DT(TIMESTR:= _NowAsTimeStruct);
END_GET
END_PROPERTY

PROPERTY NowAsTimeStruct : REFERENCE TO TIMESTRUCT
GET
NowAsTimeStruct REF= _NowAsTimeStruct;
END_GET
END_PROPERTY

END_FUNCTION_BLOCK

// ---- Classes/Edge Detection/TRisingEdge.TcPOU
FUNCTION_BLOCK TRisingEdge
VAR
    R_TRIG1 : R_TRIG;
END_VAR

PROPERTY EdgeDetected : BOOL
GET
EdgeDetected := R_TRIG1.Q;
END_GET
END_PROPERTY

METHOD Test : BOOL
VAR_INPUT
    Value : BOOL;
END_VAR
R_TRIG1(CLK := Value);
Test := R_TRIG1.Q;
END_METHOD

END_FUNCTION_BLOCK

// ---- Classes/Misc/TCounter.TcPOU
FUNCTION_BLOCK TCounter
VAR
    Count : DINT;
END_VAR

METHOD Dec : DINT
VAR_INPUT
END_VAR
Count := Count - 1;
Dec := Count;
END_METHOD

METHOD Inc : DINT
VAR_INPUT
END_VAR
Count := Count + 1;
Inc := Count;
END_METHOD

METHOD Reset
VAR_INPUT
END_VAR
Count := 0;
END_METHOD

PROPERTY Value : DINT
GET
Value := Count;
END_GET
SET
Count := Value;
END_SET
END_PROPERTY

PROPERTY ValueAsTArg : T_Arg
GET
ValueAsTArg := F_DINT(Count);
END_GET
END_PROPERTY

END_FUNCTION_BLOCK

// ---- Classes/Misc/TCsvString.TcPOU
FUNCTION_BLOCK TCsvString
VAR_INPUT
END_VAR
VAR_OUTPUT
END_VAR
VAR
    _csvString : T_MaxString;
    _FieldCount : INT;
    FieldOffsets : ARRAY[0..Param.MaxCsvFields] OF INT;
    FieldLengths : ARRAY[0..Param.MaxCsvFields] OF INT;
END_VAR

PROPERTY FieldCount : INT
GET
FieldCount := _FieldCount;
END_GET
END_PROPERTY

METHOD GetField : T_MaxString
VAR_INPUT
    Index : INT;
END_VAR
VAR
    Result : T_MaxString;
END_VAR
IF Index < _FieldCount THEN
    F_ClearMem(Result);
    MEMCPY(
        destAddr := ADR(Result),
        srcAddr  := ADR(_csvString) + INT_TO_UDINT(FieldOffsets[Index]),
        n        := INT_TO_UDINT(FieldLengths[Index]));
    GetField := Result;    
END_IF
END_METHOD

METHOD SetCsvString
VAR_INPUT
    csvString : T_MaxString;
END_VAR
VAR
    pChar : POINTER TO BYTE;
    COMMA : BYTE := F_ToASC(',');
    Fieldlength : INT;
    CharIndex : INT;
    csvStringLength : INT;
END_VAR
_csvString := csvString;
csvStringLength := LEN(_csvString);
F_ClearMem(FieldOffsets);
F_ClearMem(FieldLengths);
_FieldCount := 0;
CharIndex := 0;

IF csvStringLength > 0 THEN
    pChar := ADR(_csvString);
    
    WHILE pChar[CharIndex] <> 0 AND CharIndex < csvStringLength DO
        IF pChar[CharIndex] = COMMA THEN
            // Set length of current field...
            FieldLengths[_FieldCount] := CharIndex - FieldOffsets[_FieldCount];
            
            // Move to next field...
            IF _FieldCount < Param.MaxCsvFields - 1 THEN
                _FieldCount := _FieldCount + 1;
                // Set field offset for next field
                FieldOffsets[_FieldCount] := CharIndex + 1;
            ELSE
                EXIT;
			END_IF
		END_IF
        // Next character...
        CharIndex := CharIndex + 1;
	END_WHILE
    // no comma at end of last field...
    FieldLengths[_FieldCount] := CharIndex - FieldOffsets[_FieldCount];
    _FieldCount := _FieldCount + 1;
END_IF
END_METHOD

END_FUNCTION_BLOCK

// ---- Classes/Misc/TGetTimeZoneInfo.TcPOU
FUNCTION_BLOCK TGetTimeZoneInfo
VAR_INPUT
END_VAR
VAR_OUTPUT
END_VAR
VAR
    _Execution : TExecution;
    FB_GetTimeZoneInformation1 : FB_GetTimeZoneInformation;

    
END_VAR

FB_GetTimeZoneInformation1(
	sNetID:= , 
	bExecute:= _Execution.Starting, 
	tTimeout:= , 
	bBusy=> , 
	bError=> , 
	nErrID=> , 
	tzID=> , 
	tzInfo=> );
    
IF _Execution.Starting THEN
    _Execution.SetBusy();
END_IF

IF _Execution.Busy AND NOT FB_GetTimeZoneInformation1.bBusy THEN
    IF FB_GetTimeZoneInformation1.bError THEN
        _Execution.SetError(ErrorId := FB_GetTimeZoneInformation1.nErrID);
    ELSE
        _Execution.SetDone();
	END_IF
END_IF

PROPERTY Execution : IExecution
GET
Execution := _Execution;
END_GET
END_PROPERTY

PROPERTY TimeZoneInfo : ST_TimeZoneInformation
GET
TimeZoneInfo := FB_GetTimeZoneInformation1.tzInfo;
END_GET
END_PROPERTY

END_FUNCTION_BLOCK

// ---- Classes/Misc/TRestartTwinCAT.TcPOU
FUNCTION_BLOCK TRestartTwinCAT
VAR
    _Execution : TExecution;
    State : INT;
    StateMonitor : TValueMonitor;
    
    OnTimer : TOnTimer(Presettime := 1.0);
    TC_Restart1 : TC_Restart;
END_VAR
VAR CONSTANT
    sInit     : INT := 0;
    sDelay    : INT := 1;
    sRestart  : INT := 2;
END_VAR

StateMonitor.Test(State);
CASE State OF
    sInit:
        IF _Execution.Starting THEN
            OnTimer.Reset();
            TC_Restart1.RESTART := FALSE;
            _Execution.SetBusy();
            State := sDelay;
		END_IF
        
    sDelay:
        IF OnTimer.Run() THEN
            State := sRestart;
		END_IF
        
    sRestart:
        IF StateMonitor.Changed THEN
            TC_Restart1.RESTART := TRUE;
        ELSE
            IF NOT TC_Restart1.BUSY THEN
                IF TC_Restart1.ERR THEN
                    _Execution.SetError(ErrorId := TC_Restart1.ERRID);
                ELSE
                    _Execution.SetDone();
                END_IF
                State := sInit;
            END_IF
        END_IF
END_CASE

TC_Restart1(
	NETID:= , 
	RESTART:= , 
	TMOUT:= , 
	BUSY=> , 
	ERR=> , 
	ERRID=> );

METHOD Execute : BOOL
VAR_INPUT
    AmsNetId : T_AmsNetID;
    Delay : LREAL; // seconds
END_VAR
OnTimer.PresetTime := Delay;
TC_Restart1.NETID := AmsNetId;
Execute := _Execution.Start();
END_METHOD

PROPERTY Result : IExecutionResult
GET
Result := _Execution;
END_GET
END_PROPERTY

END_FUNCTION_BLOCK

// ---- Classes/Value Monitor/TValueMonitor.TcPOU
{attribute 'no_explicit_call':= 'do not call this POU directly'}
FUNCTION_BLOCK TValueMonitor
VAR
    _CurrentValue : INT := -1;
    _PreviousValue : INT;
    _Changed : BOOL;
END_VAR

PROPERTY Changed : BOOL
GET
Changed := _Changed;
END_GET
END_PROPERTY

PROPERTY CurrentValue : INT
GET
CurrentValue := _CurrentValue;
END_GET
END_PROPERTY

PROPERTY PreviousValue : INT
GET
PreviousValue := _PreviousValue;
END_GET
END_PROPERTY

METHOD Reset
VAR_INPUT
END_VAR
_CurrentValue := 0;
_PreviousValue := 0;
END_METHOD

METHOD Test : BOOL
VAR_INPUT
    Value : INT;
END_VAR
_Changed := Value <> _CurrentValue;
_PreviousValue := _CurrentValue;
_CurrentValue := Value;

Test := _Changed;
END_METHOD

END_FUNCTION_BLOCK

// ---- Classes/Misc/TRingCounter_INT.TcPOU
FUNCTION_BLOCK TRingCounter_INT
VAR
    Count : INT;
    _StartValue : INT;
    _EndValue : INT;
END_VAR

PROPERTY EndValue : INT
GET
EndValue := _EndValue;
END_GET
SET
_EndValue := EndValue;
END_SET
END_PROPERTY

METHOD FB_init : BOOL
VAR_INPUT
	bInitRetains : BOOL; // if TRUE, the retain variables are initialized (warm start / cold start)
	bInCopyCode : BOOL;  // if TRUE, the instance afterwards gets moved into the copy code (online change)

    StartValue : INT;
    EndValue : INT;
END_VAR
THIS^._StartValue := StartValue;
THIS^._EndValue := EndValue;
Reset();
END_METHOD

METHOD Inc
VAR_INPUT
END_VAR
Count := Count + 1;
IF Count > EndValue THEN
    Reset();
END_IF
END_METHOD

PROPERTY NextValue : INT
GET
IF Count = EndValue THEN
    NextValue := StartValue;
ELSE
    NextValue := Count + 1;
END_IF
END_GET
END_PROPERTY

METHOD Reset
VAR_INPUT
END_VAR
Count := StartValue;
END_METHOD

PROPERTY StartValue : INT
GET
StartValue := _StartValue;
END_GET
SET
_StartValue := StartValue;
END_SET
END_PROPERTY

PROPERTY Value : INT
GET
Value := Count;
END_GET
SET
Count := Value;
END_SET
END_PROPERTY

END_FUNCTION_BLOCK

// ---- Classes/Misc/TRingCounter_UDINT.TcPOU
FUNCTION_BLOCK TRingCounter_UDINT
VAR
    Count : UDINT;
    _StartValue : UDINT;
    _EndValue : UDINT;
END_VAR

PROPERTY EndValue : UDINT
GET
EndValue := _EndValue;
END_GET
SET
_EndValue := EndValue;
END_SET
END_PROPERTY

METHOD FB_init : BOOL
VAR_INPUT
	bInitRetains : BOOL; // if TRUE, the retain variables are initialized (warm start / cold start)
	bInCopyCode : BOOL;  // if TRUE, the instance afterwards gets moved into the copy code (online change)

    StartValue : UDINT;
    EndValue : UDINT;
END_VAR
THIS^._StartValue := StartValue;
THIS^._EndValue := EndValue;
Reset();
END_METHOD

METHOD Inc
VAR_INPUT
END_VAR
Count := Count + 1;
IF Count > EndValue THEN
    Reset();
END_IF
END_METHOD

PROPERTY NextValue : UDINT
GET
IF Count = EndValue THEN
    NextValue := StartValue;
ELSE
    NextValue := Count + 1;
END_IF
END_GET
END_PROPERTY

METHOD Reset
VAR_INPUT
END_VAR
Count := StartValue;
END_METHOD

PROPERTY StartValue : UDINT
GET
StartValue := _StartValue;
END_GET
SET
_StartValue := StartValue;
END_SET
END_PROPERTY

PROPERTY Value : UDINT
GET
Value := Count;
END_GET
SET
Count := Value;
END_SET
END_PROPERTY

END_FUNCTION_BLOCK

// ---- Classes/Misc/TRollingAverage.TcPOU
FUNCTION_BLOCK TRollingAverage
VAR_INPUT
END_VAR
VAR_OUTPUT
END_VAR
VAR
    pSamples : POINTER TO LREAL;
    SampleCount : UDINT;
    MaxSamples : UDINT;
END_VAR

METHOD AddSample
VAR_INPUT
    Value : LREAL;
END_VAR
IF pSamples > 0 THEN
    IF SampleCount < MaxSamples THEN
        pSamples[SampleCount] := Value;
        SampleCount := SampleCount + 1;
    ELSE
        MEMMOVE(
            destAddr := ADR(pSamples[0]),
            srcAddr  := ADR(pSamples[1]),
            n        := SIZEOF(pSamples[0]) * (MaxSamples-1));
        pSamples[MaxSamples - 1] := Value;
    END_IF
END_IF
END_METHOD

METHOD Clear
VAR_INPUT
END_VAR
IF pSamples > 0 THEN
    MEMSET(
        destAddr := pSamples,
        fillByte := 0,
        n        := MaxSamples * SIZEOF(pSamples[0]));
        
    SampleCount := 0;
END_IF
END_METHOD

METHOD FB_exit : BOOL
VAR_INPUT
	bInCopyCode : BOOL; // if TRUE, the exit method is called for exiting an instance that is copied afterwards (online change).
END_VAR
IF bInCopyCode = FALSE THEN // avoid deleting samples on online change!
    __DELETE(pSamples);
END_IF
END_METHOD

METHOD FB_init : BOOL
VAR_INPUT
	bInitRetains : BOOL; // if TRUE, the retain variables are initialized (warm start / cold start)
	bInCopyCode : BOOL;  // if TRUE, the instance afterwards gets moved into the copy code (online change)
    MaxSamples : UDINT;
END_VAR
pSamples := __NEW(LREAL,MaxSamples);
THIS^.MaxSamples := MaxSamples;
END_METHOD

METHOD GetAverage : LREAL
VAR
    i : UDINT;
    Sum : LREAL;
END_VAR
IF pSamples > 0 AND SampleCount > 0 THEN
    FOR i := 0 TO SampleCount - 1 DO
        Sum := Sum + pSamples[i];
    END_FOR
    GetAverage := Sum/SampleCount;
END_IF
END_METHOD

END_FUNCTION_BLOCK

// ---- Classes/Misc/TSetWindowsClock.TcPOU
FUNCTION_BLOCK TSetWindowsClock
VAR
    Execution : TExecution;
    NT_SetLocalTime1 : NT_SetLocalTime;
END_VAR

NT_SetLocalTime1(
	NETID:= , 
	TIMESTR:= , 
	START:= Execution.Starting, 
	TMOUT:= , 
	BUSY=> , 
	ERR=> , 
	ERRID=> );
    
IF Execution.Starting THEN
    Execution.SetBusy();
END_IF

IF Execution.Busy AND NOT NT_SetLocalTime1.BUSY THEN
    IF NT_SetLocalTime1.ERR THEN
        Execution.SetError(ErrorId := NT_SetLocalTime1.ERRID);
    ELSE
        Execution.SetDone();
	END_IF
END_IF

METHOD Execute : BOOL
VAR_INPUT
    AmsNetId : T_AmsNetID;
    TimeStruct : TimeStruct;
END_VAR
IF Execution.Start() THEN
    NT_SetLocalTime1.TIMESTR := TimeStruct;
    NT_SetLocalTime1.NETID := AmsNetId;
    Execute := TRUE;
END_IF
END_METHOD

PROPERTY ExecutionResult  : IExecutionResult
GET
ExecutionResult := Execution;
END_GET
END_PROPERTY

END_FUNCTION_BLOCK

// ---- Classes/Misc/TShutdown.TcPOU
FUNCTION_BLOCK TShutdown
VAR
    _Execution : TExecution;
    NT_Shutdown1 : NT_Shutdown;
END_VAR

NT_Shutdown1(
	NETID:= , 
	DELAY:= , 
	START:= _Execution.Starting, 
	TMOUT:= , 
	BUSY=> , 
	ERR=> , 
	ERRID=> );

IF _Execution.Starting THEN
    _Execution.SetBusy();
END_IF

IF _Execution.Busy AND NOT NT_Shutdown1.BUSY THEN
    IF NT_Shutdown1.ERR THEN
        _Execution.SetError(ErrorId := NT_Shutdown1.ERRID);
    ELSE
        _Execution.SetDone();
	END_IF
END_IF

METHOD Execute : BOOL
VAR_INPUT
    AmsNetId : T_AmsNetID;
    Delay : DWORD;
END_VAR
NT_Shutdown1.DELAY := Delay;


NT_Shutdown1.NETID := AmsNetId;
Execute := _Execution.Start();
END_METHOD

PROPERTY Result : IExecutionResult
GET
Result := _Execution;
END_GET
END_PROPERTY

END_FUNCTION_BLOCK

// ---- Classes/Misc/TStartProcess.TcPOU
FUNCTION_BLOCK TStartProcess
VAR
    _Execution : TExecution;
    NT_StartProcess1 : NT_StartProcess;
END_VAR

NT_StartProcess1(
	NETID:= , 
	PATHSTR:= , 
	DIRNAME:= , 
	COMNDLINE:= , 
	START:= _Execution.Starting, 
	TMOUT:= , 
	BUSY=> , 
	ERR=> , 
	ERRID=> );
    
IF _Execution.Starting THEN
    _Execution.SetBusy();
END_IF

IF _Execution.Busy AND NOT NT_StartProcess1.BUSY THEN
    IF NT_StartProcess1.ERR THEN
        _Execution.SetError(ErrorId := NT_StartProcess1.ERRID);
    ELSE
        _Execution.SetDone();
	END_IF
END_IF

METHOD Execute : BOOL
VAR_INPUT
    AmsNetId : T_AmsNetID;
    Directory : T_MaxString;
    Path : T_MaxString;
END_VAR
NT_StartProcess1.DIRNAME := Directory;
NT_StartProcess1.PATHSTR := Path;
NT_StartProcess1.NETID := AmsNetId;
Execute := _Execution.Start();
END_METHOD

PROPERTY Result : IExecutionResult
GET
Result := _Execution;
END_GET
END_PROPERTY

END_FUNCTION_BLOCK

// ---- Classes/Timers/TPulseTimer.TcPOU
FUNCTION_BLOCK TPulseTimer
VAR
    TP1 : TP;
END_VAR

METHOD FB_init : BOOL
VAR_INPUT
	bInitRetains : BOOL; // if TRUE, the retain variables are initialized (warm start / cold start)
	bInCopyCode : BOOL;  // if TRUE, the instance afterwards gets moved into the copy code (online change)
    PresetTime : LREAL; // seconds
END_VAR
TP1.PT := LREAL_TO_TIME(PresetTime * 1000);
END_METHOD

PROPERTY OutputState : BOOL
GET
OutputState := TP1.Q;
END_GET
END_PROPERTY

PROPERTY PresetTime : LREAL
GET
PresetTime := TIME_TO_LREAL(TP1.PT)/1000.0; // in seconds
END_GET
SET
TP1.PT := LREAL_TO_TIME(PresetTime * 1000);
END_SET
END_PROPERTY

METHOD Pulse : BOOL
VAR_INPUT
    In : BOOL;
END_VAR
TP1(IN := In);
Pulse := TP1.Q;
END_METHOD

METHOD Reset
TP1(IN := FALSE);
END_METHOD

METHOD Run : BOOL
TP1(IN := TRUE);
Run := TP1.Q;
END_METHOD

END_FUNCTION_BLOCK

// ---- Classes/Value Monitor/TValueMonitorEx.TcPOU
{attribute 'no_explicit_call':= 'do not call this POU directly'}
FUNCTION_BLOCK TValueMonitorEx
VAR
    _Changed : BOOL;
    StoredValue : ARRAY[0..7] OF BYTE;
END_VAR

PROPERTY Changed : BOOL
GET
Changed := _Changed;
END_GET
END_PROPERTY

METHOD Reset
VAR_INPUT
END_VAR
MEMSET(
    destAddr := ADR(StoredValue),
    fillByte  := 16#00,
    n        := SIZEOF(StoredValue));
END_METHOD

METHOD Test : BOOL;
VAR_INPUT
    Value : ANY;
END_VAR
_Changed := 0 <>  MEMCMP(
                    pBuf1 := Value.pValue,
                    pBuf2 := ADR(StoredValue),
                    n     := DINT_TO_UDINT(Value.diSize));
    
IF _Changed THEN
    MEMCPY(
        destAddr := ADR(StoredValue),
        srcAddr  := Value.pValue,
        n        := DINT_TO_UDINT(Value.diSize));
END_IF

Test := _Changed;
END_METHOD

END_FUNCTION_BLOCK

// ---- Function Blocks/FB_AutoReset.TcPOU
FUNCTION_BLOCK FB_AutoReset
// Automatically resets the boolean Value after the time period
VAR_INPUT
    Value : REFERENCE TO BOOL;
    PT : TIME;
END_VAR
VAR
    TON1 : TON;
END_VAR

TON1(IN := Value, PT := PT);
IF TON1.Q THEN
    Value := FALSE;
END_IF

END_FUNCTION_BLOCK

// ---- Function Blocks/FB_ValueChanged.TcPOU
FUNCTION_BLOCK FB_ValueChanged
VAR_INPUT
    Value : INT;
END_VAR
VAR_OUTPUT
    Changed : BOOL;
END_VAR
VAR
    OldValue : INT;
END_VAR

Changed := Value <> OldValue;
OldValue := Value;

END_FUNCTION_BLOCK

// ---- Functions/Event Logging/F_LogMessage.TcPOU
FUNCTION F_LogMessage : T_MaxString
VAR_INPUT
    Source  : T_MaxString;
    Message : T_MaxString;
END_VAR

ADSLOGSTR(
    msgCtrlMask := ADSLOG_MSGTYPE_STRING OR ADSLOG_MSGTYPE_HINT OR ADSLOG_MSGTYPE_LOG,
    msgFmtStr := F_FormatStringEx2('%s : %s',Source,Message),
    strArg := '');

END_FUNCTION

// ---- Functions/Event Logging/F_LogWarning.TcPOU
FUNCTION F_LogWarning : T_MaxString 
VAR_INPUT
    Source  : T_MaxString;
    Message : T_MaxString;
END_VAR

ADSLOGSTR(
    msgCtrlMask := ADSLOG_MSGTYPE_STRING OR ADSLOG_MSGTYPE_WARN OR ADSLOG_MSGTYPE_LOG,
    msgFmtStr := F_FormatStringEx2('%s : %s',Source,Message),
    strArg := '');

END_FUNCTION

// ---- Functions/String Formatting/F_FormatString5.TcPOU
FUNCTION F_FormatString5 : T_MaxString
VAR_INPUT
	Format	: T_MaxString;
	arg1	: T_Arg;
	arg2	: T_Arg;
	arg3	: T_Arg;
	arg4	: T_Arg;
	arg5	: T_Arg;
END_VAR
VAR
    FB_FormatString1 : FB_FormatString;
END_VAR

FB_FormatString1(
	sFormat:= Format, 
	arg1:= arg1, 
	arg2:= arg2, 
	arg3:= arg3, 
	arg4:= arg4, 
	arg5:= arg5, 
	arg6:= , 
	arg7:= , 
	arg8:= , 
	arg9:= , 
	arg10:= , 
	bError=> , 
	nErrId=> , 
	sOut=> F_FormatString5);

END_FUNCTION

// ---- Functions/String Formatting/F_FormatStringEx10.TcPOU
FUNCTION F_FormatStringEx10 : T_MaxString
VAR_INPUT
	Format	: T_MaxString;
	arg1	: T_MaxString;
	arg2	: T_MaxString;
	arg3	: T_MaxString;
	arg4	: T_MaxString;
	arg5	: T_MaxString;
	arg6	: T_MaxString;
	arg7	: T_MaxString;
	arg8	: T_MaxString;
	arg9	: T_MaxString;
	arg10	: T_MaxString;
END_VAR
VAR
    FB_FormatString1 : FB_FormatString;
END_VAR



FB_FormatString1(
	sFormat:= Format, 
	arg1 := F_STRING(arg1), 
	arg2 := F_STRING(arg2),
	arg3 := F_STRING(arg3), 
	arg4 := F_STRING(arg4), 
	arg5 := F_STRING(arg5), 
	arg6 := F_STRING(arg6), 
	arg7 := F_STRING(arg7), 
	arg8 := F_STRING(arg8),  
	arg9 := F_STRING(arg9), 
	arg10:= F_STRING(arg10), 
	bError=> , 
	nErrId=> , 
	sOut=> F_FormatStringEx10);

END_FUNCTION

// ---- Functions/String Formatting/F_FormatStringEx6.TcPOU
FUNCTION F_FormatStringEx6 : T_MaxString
VAR_INPUT
	Format	: T_MaxString;
	arg1	: T_MaxString;
	arg2	: T_MaxString;
	arg3	: T_MaxString;
	arg4	: T_MaxString;
	arg5	: T_MaxString;
	arg6	: T_MaxString;
END_VAR
VAR
    FB_FormatString1 : FB_FormatString;
END_VAR



FB_FormatString1(
	sFormat:= Format, 
	arg1:= F_STRING(arg1), 
	arg2:= F_STRING(arg2),
	arg3:= F_STRING(arg3), 
	arg4:= F_STRING(arg4), 
	arg5:= F_STRING(arg5), 
	arg6:= F_STRING(arg6), 
	arg7:= , 
	arg8:= , 
	arg9:= , 
	arg10:= , 
	bError=> , 
	nErrId=> , 
	sOut=> F_FormatStringEx6);

END_FUNCTION

// ---- Functions/String Formatting/F_FormatStringEx8.TcPOU
FUNCTION F_FormatStringEx8 : T_MaxString
VAR_INPUT
	Format	: T_MaxString;
	arg1	: T_MaxString;
	arg2	: T_MaxString;
	arg3	: T_MaxString;
	arg4	: T_MaxString;
	arg5	: T_MaxString;
	arg6	: T_MaxString;
	arg7	: T_MaxString;
	arg8	: T_MaxString;
END_VAR
VAR
    FB_FormatString1 : FB_FormatString;
END_VAR



FB_FormatString1(
	sFormat:= Format, 
	arg1:= F_STRING(arg1), 
	arg2:= F_STRING(arg2),
	arg3:= F_STRING(arg3), 
	arg4:= F_STRING(arg4), 
	arg5:= F_STRING(arg5), 
	arg6:= F_STRING(arg6), 
	arg7:= F_STRING(arg7), 
	arg8:= F_STRING(arg8),  
	arg9:= , 
	arg10:= , 
	bError=> , 
	nErrId=> , 
	sOut=> F_FormatStringEx8);

END_FUNCTION

// ---- Functions/String Formatting/F_PadString.TcPOU
FUNCTION F_PadString : T_MaxString // pad string with spaces or trim from rhs to fix length of string
VAR_INPUT
    InputString : T_MaxString;
    Length : UINT;
END_VAR
VAR
    InputStringLength : UINT;
    Result : T_MaxString;
    TrimLength : UINT;
    PaddingLength : UINT;
    i : UINT;
END_VAR

InputStringLength := INT_TO_UINT(MAX(0,LEN(InputString)));
Result := InputString;

IF InputStringLength > Length THEN
    TrimLength := InputStringLength - Length;
    Result := F_RTrimEx(TrimLength,Result);
    
ELSIF InputStringLength < Length THEN
    PaddingLength := Length - InputStringLength;

    FOR i := 1 TO PaddingLength DO
        Result := CONCAT(Result,' ');
	END_FOR
    
END_IF

F_PadString := Result;

END_FUNCTION

// ---- Functions/String Formatting/F_RTrimEx.TcPOU
FUNCTION F_RTrimEx : T_MaxString // removes n characters from end of string
VAR_INPUT
   n : UINT; 
   str : T_MaxString;
END_VAR
VAR
    Length : UINT;
END_VAR

Length := INT_TO_UINT(LEN(str));
IF n > 0 AND n < Length THEN
    // overwrite chars to be trimmed with nulls...
    MEMSET(destAddr := ADR(str) + Length - n,
           fillByte:= 0,
           n := n); 
    
END_IF
F_RTrimEx := str;

END_FUNCTION

// ---- Visualisation/Visualization.TcVIS
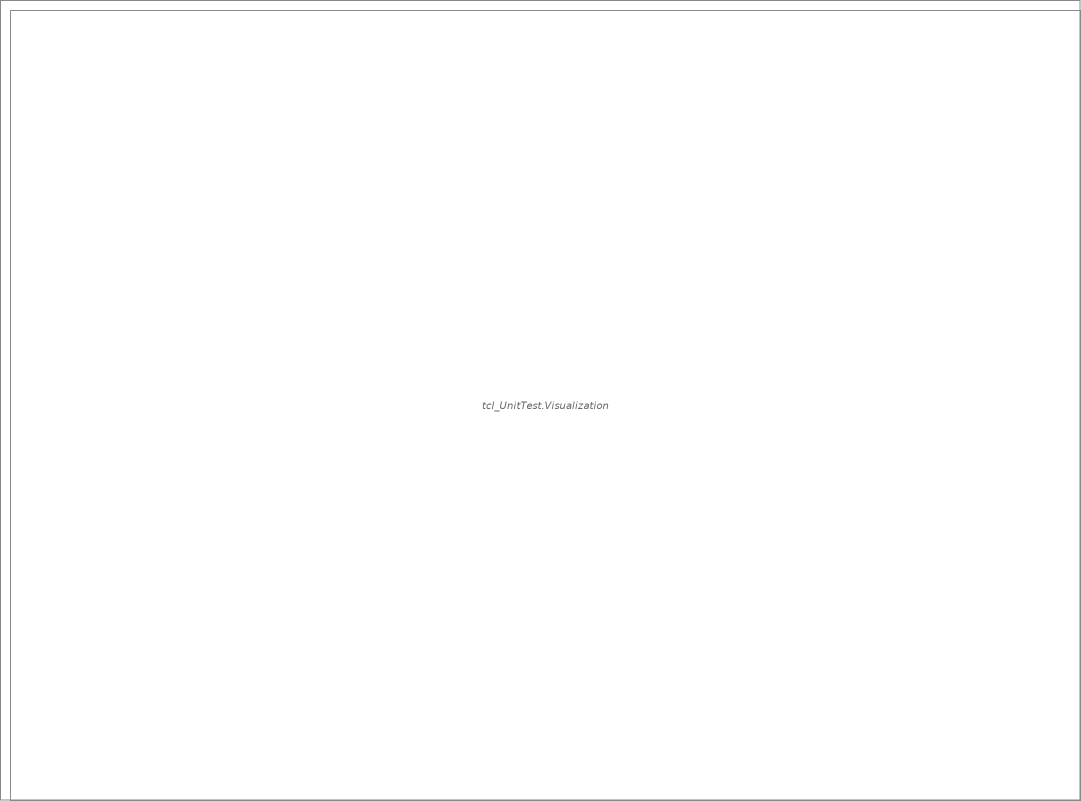
VISUALIZATION Visualization  // 1081x801
    Frame (10,10 1071x791)
        shows tcl_UnitTest.Visualization()
END_VISUALIZATION
